// TIA Portal V17 export
// export: Created 2023-12-22T15:03:07.6064327Z, ExportSetting WithDefaults, DisplayName Totally Integrated Automation Portal, DisplayVersion V17, DisplayName TIA Portal Openness, DisplayVersion V17, DisplayName TIA Portal Version Control Interface, DisplayVersion V17, DisplayName STEP 7 Professional, DisplayVersion V17, DisplayName STEP 7 Safety, DisplayVersion V17, DisplayName WinCC Advanced, DisplayVersion V17
FUNCTION_BLOCK "ModBus_TCP"   // FB40, LAD
TITLE = Блок опроса ModBus TCP
{ S7_Optimized_Access := 'FALSE' }
VERSION : 0.1
// ВНИМАНИЕ!  Через один аппаратный порт контроллера можно проводить множество различных опросов по ModBus TCP. Для этого у каждого экземпляра должен быть указан уникальный CONNECT.ID.
// 
// Для каждого уникального CONNECT.ID / внешней ветки / точки подключения (IP, RemotePort) рекомендуется использовать отдельный экземпляр функционального блока. Например, при использовании tGW-735 имеющего 3 порта подключения с RemotePort = 502, 503 и 504 соответственно (но общий IP адрес) рекомендуется использовать три отдельных блока ModBus_TCP с уникальными CONNECT.ID.
// 
// Каждая точка чтения/записи = 1 экземпляр DEV_Config, количество элементов в массиве можно менять по необходимости, итоговое количество элементов массива указывается в теге Limit.
// 
// Для режима чтения необходимо указать:
// - MODE = 0
// - Source_DB = 40 (номер DB Modbus_TCP_DB)
// - SourceOFFSET = 0
// - Target_DB = xx (номер DB, куда необходимо положить прочитанные данные)
// - Target_OFFSET = xx (номер байта, начиная с которого кладутся прочитанные данные в выбранный DB)
// 
// Для режима опроса необходимо указать:
// - MODE = 1
// - Source_DB = xx (номер DB, откуда необходимо взять данные для передачи)
// - Source_OFFSET = xx (номер байта, начиная с которого берутся данные для передачи)
// - Target_DB = 40 (номер DB Modbus_TCP_DB)
// - Target_OFFSET = 0
// stored: AutoNumber false, IsIECCheckEnabled false, SetENOAutomatically false, UDAEnableTagReadback false
   VAR DB_SPECIFIC
      DATA : Array[0..100] of Word;   // Массив данных
      CONNECT { S7_SetPoint := 'True'} : TCON_IP_v4;
   END_VAR
   // CONNECT.InterfaceId := 64;
   // CONNECT.ID := 16#0001;
   // CONNECT.ConnectionType := 16#0B;
   // CONNECT.ActiveEstablished := TRUE;
   // CONNECT.RemoteAddress.ADDR[1] := 16#C0;
   // CONNECT.RemoteAddress.ADDR[2] := 16#A8;
   // CONNECT.RemoteAddress.ADDR[3] := 16#00;
   // CONNECT.RemoteAddress.ADDR[4] := 16#0A;
   // CONNECT.RemotePort := 502;
   // CONNECT.LocalPort := 0;
BEGIN

REGION Network 1
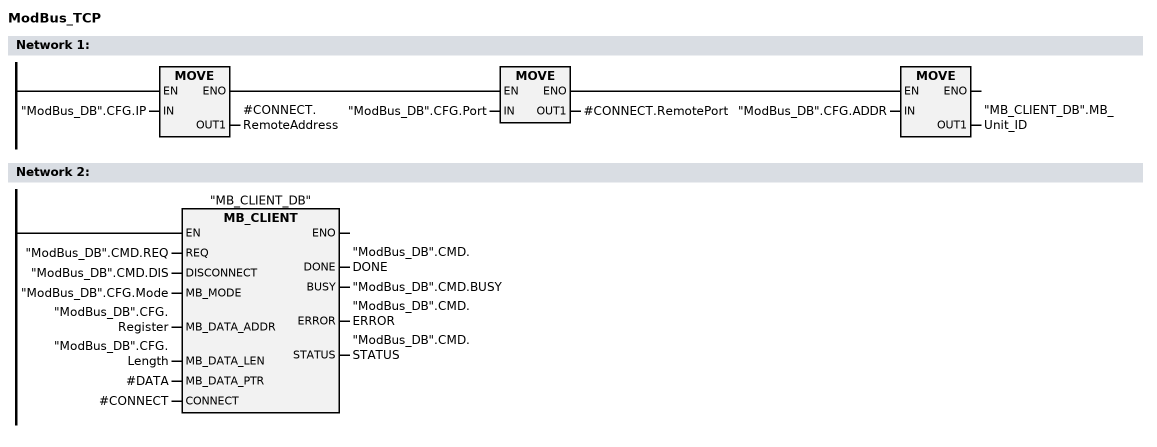
   RUNG wire#powerrail
      Move(in := "ModBus_DB".CFG.IP, out1 => #CONNECT.RemoteAddress)
      Move(in := "ModBus_DB".CFG.Port, out1 => #CONNECT.RemotePort)
      Move(in := "ModBus_DB".CFG.ADDR, out1 => "MB_CLIENT_DB".MB_Unit_ID)
   END_RUNG
   // the same network as SCL:
   #CONNECT.RemoteAddress := "ModBus_DB".CFG.IP;
   #CONNECT.RemotePort := "ModBus_DB".CFG.Port;
   "MB_CLIENT_DB".MB_Unit_ID := "ModBus_DB".CFG.ADDR;
END_REGION

REGION Network 2
   RUNG wire#powerrail
      "MB_CLIENT_DB".MB_CLIENT(REQ := "ModBus_DB".CMD.REQ, DISCONNECT := "ModBus_DB".CMD.DIS, MB_MODE := "ModBus_DB".CFG.Mode, MB_DATA_ADDR := "ModBus_DB".CFG.Register, MB_DATA_LEN := "ModBus_DB".CFG.Length, MB_DATA_PTR := #DATA, CONNECT := #CONNECT, DONE => "ModBus_DB".CMD.DONE, BUSY => "ModBus_DB".CMD.BUSY, ERROR => "ModBus_DB".CMD.ERROR, STATUS => "ModBus_DB".CMD.STATUS)
   END_RUNG
   // the same network as SCL:
   "MB_CLIENT_DB"(REQ := "ModBus_DB".CMD.REQ,   // MB_CLIENT
                  DISCONNECT := "ModBus_DB".CMD.DIS,
                  MB_MODE := "ModBus_DB".CFG.Mode,
                  MB_DATA_ADDR := "ModBus_DB".CFG.Register,
                  MB_DATA_LEN := "ModBus_DB".CFG.Length,
                  MB_DATA_PTR := #DATA,
                  CONNECT := #CONNECT,
                  DONE => "ModBus_DB".CMD.DONE,
                  BUSY => "ModBus_DB".CMD.BUSY,
                  ERROR => "ModBus_DB".CMD.ERROR,
                  STATUS => "ModBus_DB".CMD.STATUS);
END_REGION
END_FUNCTION_BLOCK
